PROGRAM SafetyMode
VAR
	
END_VAR

IF RunTCP.sCommand = 'HIGHMODE' THEN
	GVL_SAFETY.LowMode := FALSE;
ELSIF RunTCP.sCommand = 'LOWMODE' THEN
	GVL_SAFETY.LowMode := TRUE;
END_IF

END_PROGRAM

(* stored: Version 1.1.0.1, ProductVersion 3.1.4024.3
   POU SafetyMode: Id {f3338e28-180f-4591-ab90-39c1de9b87e9}, SpecialFunc None *)
